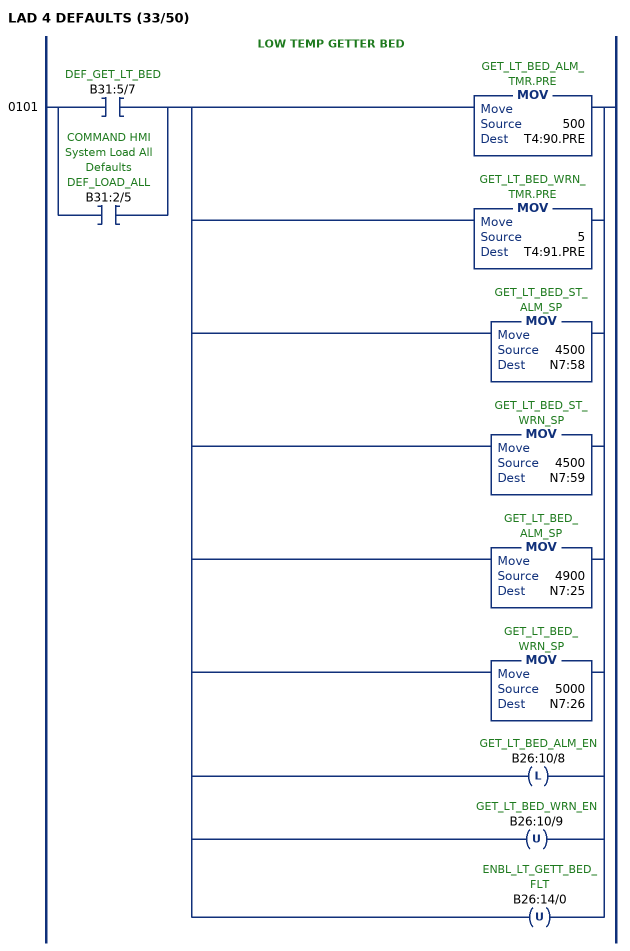
% Rung: 101 %
% TITLE: LOW TEMP GETTER BED %
SOR BST XIC B31:5/7 NXB XIC B31:2/5 BND BST MOV 500 T4:90.PRE NXB MOV 5 T4:91.PRE NXB BST MOV 4500 N7:58 NXB MOV 4500 N7:59 BND NXB BST MOV 4900 N7:25 NXB MOV 5000 N7:26 BND NXB OTL B26:10/8 NXB OTU B26:10/9 NXB OTU B26:14/0 BND EOR
%   B31:5/7  DEF_GET_LT_BED %
%   B31:2/5  DEF_LOAD_ALL  "COMMAND HMI System Load All Defaults" %
%   T4:90  GET_LT_BED_ALM_TMR %
%   T4:91  GET_LT_BED_WRN_TMR %
%   N7:58  GET_LT_BED_ST_ALM_SP %
%   N7:59  GET_LT_BED_ST_WRN_SP %
%   N7:25  GET_LT_BED_ALM_SP %
%   N7:26  GET_LT_BED_WRN_SP %
%   B26:10/8  GET_LT_BED_ALM_EN %
%   B26:10/9  GET_LT_BED_WRN_EN %
%   B26:14/0  ENBL_LT_GETT_BED_FLT %

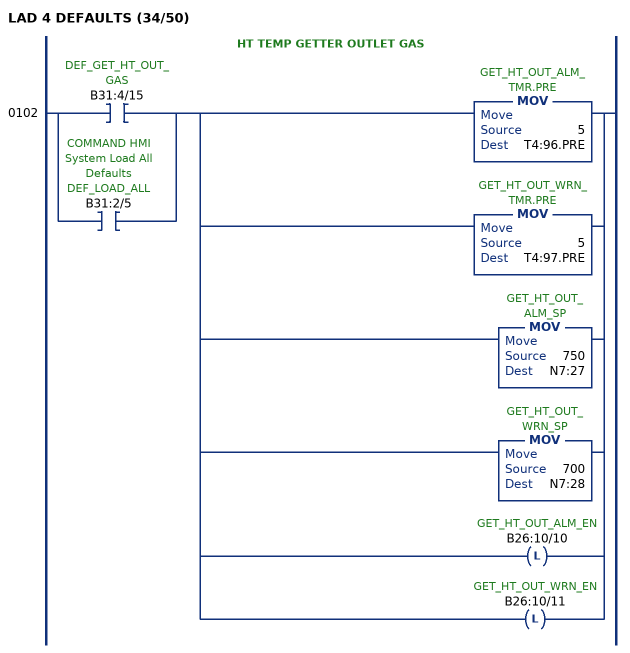
% Rung: 102 %
% TITLE: HT TEMP GETTER OUTLET GAS %
SOR BST XIC B31:4/15 NXB XIC B31:2/5 BND BST MOV 5 T4:96.PRE NXB MOV 5 T4:97.PRE NXB MOV 750 N7:27 NXB MOV 700 N7:28 NXB OTL B26:10/10 NXB OTL B26:10/11 BND EOR
%   B31:4/15  DEF_GET_HT_OUT_GAS %
%   B31:2/5  DEF_LOAD_ALL  "COMMAND HMI System Load All Defaults" %
%   T4:96  GET_HT_OUT_ALM_TMR %
%   T4:97  GET_HT_OUT_WRN_TMR %
%   N7:27  GET_HT_OUT_ALM_SP %
%   N7:28  GET_HT_OUT_WRN_SP %
%   B26:10/10  GET_HT_OUT_ALM_EN %
%   B26:10/11  GET_HT_OUT_WRN_EN %

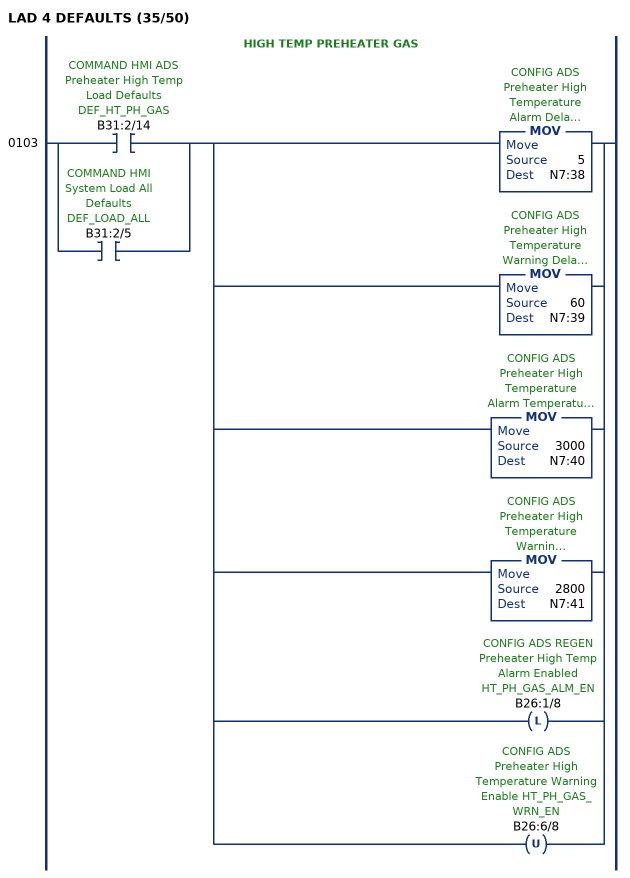
% Rung: 103 %
% TITLE: HIGH TEMP PREHEATER GAS %
SOR BST XIC B31:2/14 NXB XIC B31:2/5 BND BST MOV 5 N7:38 NXB MOV 60 N7:39 NXB MOV 3000 N7:40 NXB MOV 2800 N7:41 NXB OTL B26:1/8 NXB OTU B26:6/8 BND EOR
%   B31:2/14  DEF_HT_PH_GAS  "COMMAND HMI ADS Preheater High Temp Load Defaults" %
%   B31:2/5  DEF_LOAD_ALL  "COMMAND HMI System Load All Defaults" %
%   N7:38  HT_PH_GAS_ALM_DLY  "CONFIG ADS Preheater High Temperature Alarm Delay" %
%   N7:39  HT_PH_GAS_WRN_DLY  "CONFIG ADS Preheater High Temperature Warning Delay" %
%   N7:40  HT_PH_GAS_ALM_SP  "CONFIG ADS Preheater High Temperature Alarm Temperature" %
%   N7:41  HT_PH_GAS_WRN_SP  "CONFIG ADS Preheater High Temperature Warning Temperature" %
%   B26:1/8  HT_PH_GAS_ALM_EN  "CONFIG ADS REGEN Preheater High Temp Alarm Enabled" %
%   B26:6/8  HT_PH_GAS_WRN_EN  "CONFIG ADS Preheater High Temperature Warning Enable" %

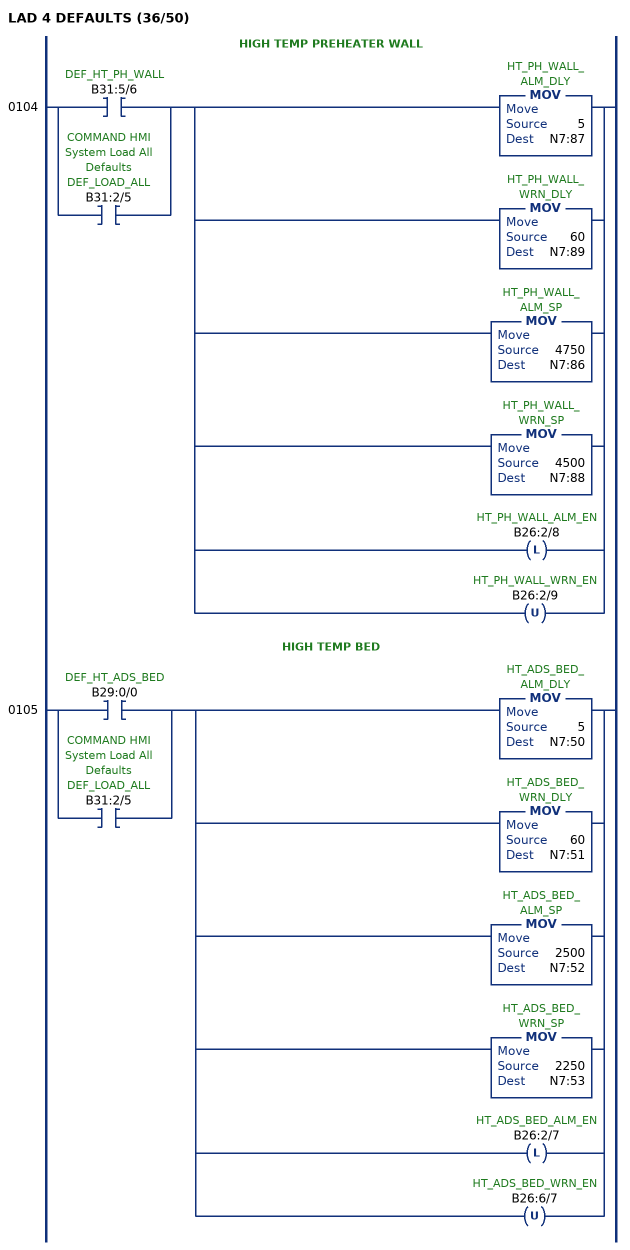
% Rung: 104 %
% TITLE: HIGH TEMP PREHEATER WALL %
SOR BST XIC B31:5/6 NXB XIC B31:2/5 BND BST MOV 5 N7:87 NXB MOV 60 N7:89 NXB MOV 4750 N7:86 NXB MOV 4500 N7:88 NXB OTL B26:2/8 NXB OTU B26:2/9 BND EOR
%   B31:5/6  DEF_HT_PH_WALL %
%   B31:2/5  DEF_LOAD_ALL  "COMMAND HMI System Load All Defaults" %
%   N7:87  HT_PH_WALL_ALM_DLY %
%   N7:89  HT_PH_WALL_WRN_DLY %
%   N7:86  HT_PH_WALL_ALM_SP %
%   N7:88  HT_PH_WALL_WRN_SP %
%   B26:2/8  HT_PH_WALL_ALM_EN %
%   B26:2/9  HT_PH_WALL_WRN_EN %
% Rung: 105 %
% TITLE: HIGH TEMP BED %
SOR BST XIC B29:0/0 NXB XIC B31:2/5 BND BST MOV 5 N7:50 NXB MOV 60 N7:51 NXB MOV 2500 N7:52 NXB MOV 2250 N7:53 NXB OTL B26:2/7 NXB OTU B26:6/7 BND EOR
%   B29:0/0  DEF_HT_ADS_BED %
%   B31:2/5  DEF_LOAD_ALL  "COMMAND HMI System Load All Defaults" %
%   N7:50  HT_ADS_BED_ALM_DLY %
%   N7:51  HT_ADS_BED_WRN_DLY %
%   N7:52  HT_ADS_BED_ALM_SP %
%   N7:53  HT_ADS_BED_WRN_SP %
%   B26:2/7  HT_ADS_BED_ALM_EN %
%   B26:6/7  HT_ADS_BED_WRN_EN %

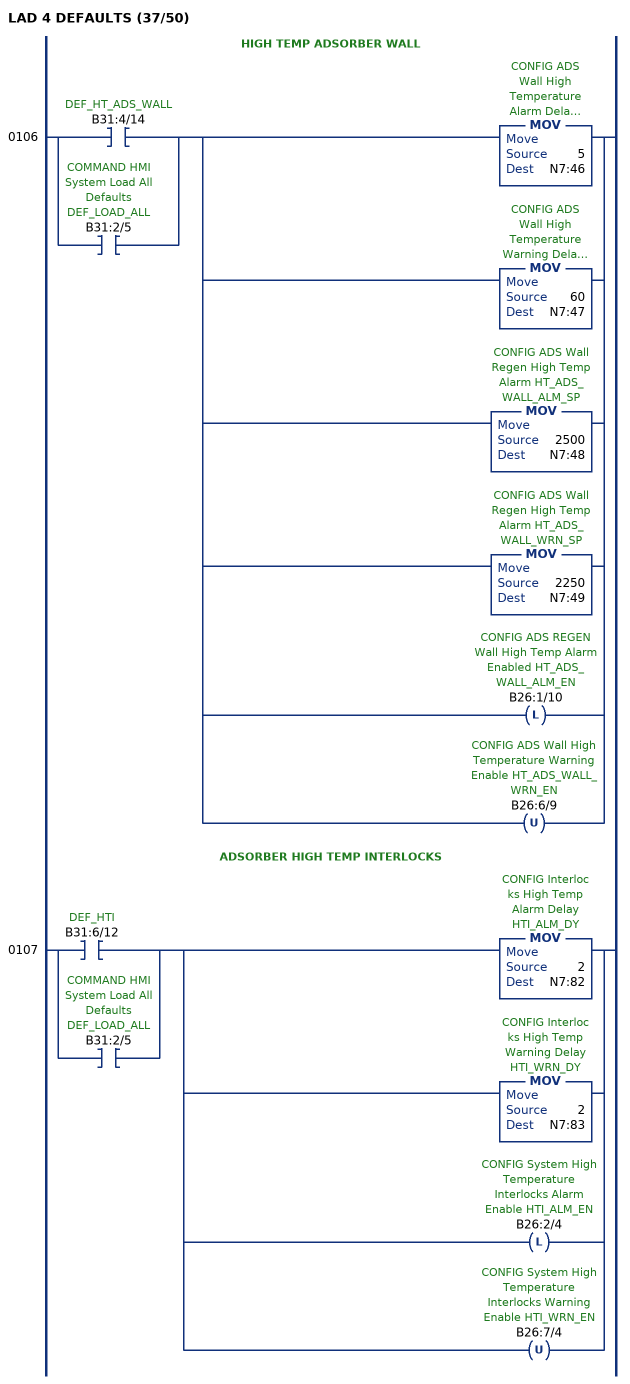
% Rung: 106 %
% TITLE: HIGH TEMP ADSORBER WALL %
SOR BST XIC B31:4/14 NXB XIC B31:2/5 BND BST MOV 5 N7:46 NXB MOV 60 N7:47 NXB MOV 2500 N7:48 NXB MOV 2250 N7:49 NXB OTL B26:1/10 NXB OTU B26:6/9 BND EOR
%   B31:4/14  DEF_HT_ADS_WALL %
%   B31:2/5  DEF_LOAD_ALL  "COMMAND HMI System Load All Defaults" %
%   N7:46  HT_ADS_WALL_ALM_DLY  "CONFIG ADS Wall High Temperature Alarm Delay" %
%   N7:47  HT_ADS_WALL_WRN_DLY  "CONFIG ADS Wall High Temperature Warning Delay" %
%   N7:48  HT_ADS_WALL_ALM_SP  "CONFIG ADS Wall Regen High Temp Alarm" %
%   N7:49  HT_ADS_WALL_WRN_SP  "CONFIG ADS Wall Regen High Temp Alarm" %
%   B26:1/10  HT_ADS_WALL_ALM_EN  "CONFIG ADS REGEN Wall High Temp Alarm Enabled" %
%   B26:6/9  HT_ADS_WALL_WRN_EN  "CONFIG ADS Wall High Temperature Warning Enable" %
% Rung: 107 %
% TITLE: ADSORBER HIGH TEMP INTERLOCKS %
SOR BST XIC B31:6/12 NXB XIC B31:2/5 BND BST MOV 2 N7:82 NXB MOV 2 N7:83 NXB OTL B26:2/4 NXB OTU B26:7/4 BND EOR
%   B31:6/12  DEF_HTI %
%   B31:2/5  DEF_LOAD_ALL  "COMMAND HMI System Load All Defaults" %
%   N7:82  HTI_ALM_DY  "CONFIG Interlocks High Temp Alarm Delay" %
%   N7:83  HTI_WRN_DY  "CONFIG Interlocks High Temp Warning Delay" %
%   B26:2/4  HTI_ALM_EN  "CONFIG System High Temperature Interlocks Alarm Enable" %
%   B26:7/4  HTI_WRN_EN  "CONFIG System High Temperature Interlocks Warning Enable" %

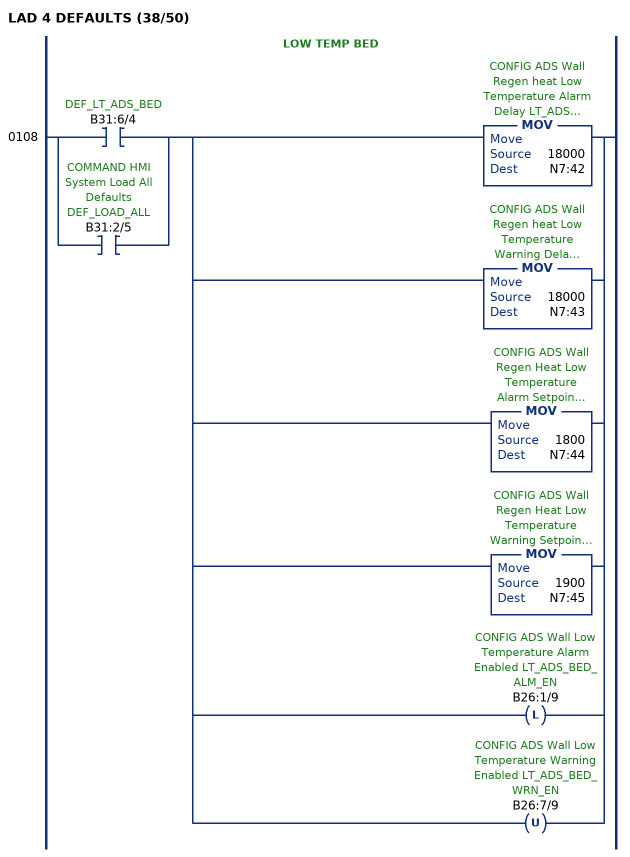
% Rung: 108 %
% TITLE: LOW TEMP BED %
SOR BST XIC B31:6/4 NXB XIC B31:2/5 BND BST MOV 18000 N7:42 NXB MOV 18000 N7:43 NXB MOV 1800 N7:44 NXB MOV 1900 N7:45 NXB OTL B26:1/9 NXB OTU B26:7/9 BND EOR
%   B31:6/4  DEF_LT_ADS_BED %
%   B31:2/5  DEF_LOAD_ALL  "COMMAND HMI System Load All Defaults" %
%   N7:42  LT_ADS_BED_ALM_DLY  "CONFIG ADS Wall Regen heat Low Temperature Alarm Delay" %
%   N7:43  LT_ADS_BED_WRN_DLY  "CONFIG ADS Wall Regen heat Low Temperature Warning Delay" %
%   N7:44  LT_ADS_BED_ALM_SP  "CONFIG ADS Wall Regen Heat Low Temperature Alarm Setpoint" %
%   N7:45  LT_ADS_BED_WRN_SP  "CONFIG ADS Wall Regen Heat Low Temperature Warning Setpoint" %
%   B26:1/9  LT_ADS_BED_ALM_EN  "CONFIG ADS Wall Low Temperature Alarm Enabled" %
%   B26:7/9  LT_ADS_BED_WRN_EN  "CONFIG ADS Wall Low Temperature Warning Enabled" %

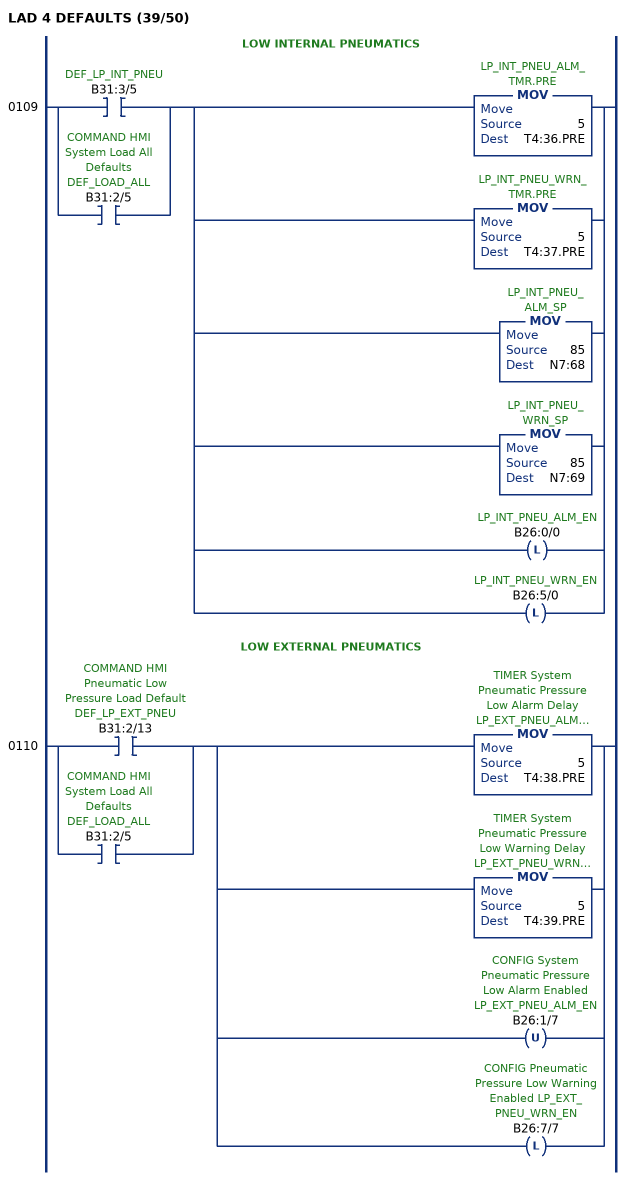
% Rung: 109 %
% TITLE: LOW INTERNAL PNEUMATICS %
SOR BST XIC B31:3/5 NXB XIC B31:2/5 BND BST MOV 5 T4:36.PRE NXB MOV 5 T4:37.PRE NXB MOV 85 N7:68 NXB MOV 85 N7:69 NXB OTL B26:0/0 NXB OTL B26:5/0 BND EOR
%   B31:3/5  DEF_LP_INT_PNEU %
%   B31:2/5  DEF_LOAD_ALL  "COMMAND HMI System Load All Defaults" %
%   T4:36  LP_INT_PNEU_ALM_TMR %
%   T4:37  LP_INT_PNEU_WRN_TMR %
%   N7:68  LP_INT_PNEU_ALM_SP %
%   N7:69  LP_INT_PNEU_WRN_SP %
%   B26:0/0  LP_INT_PNEU_ALM_EN %
%   B26:5/0  LP_INT_PNEU_WRN_EN %
% Rung: 110 %
% TITLE: LOW EXTERNAL PNEUMATICS %
SOR BST XIC B31:2/13 NXB XIC B31:2/5 BND BST MOV 5 T4:38.PRE NXB MOV 5 T4:39.PRE NXB OTU B26:1/7 NXB OTL B26:7/7 BND EOR
%   B31:2/13  DEF_LP_EXT_PNEU  "COMMAND HMI Pneumatic Low Pressure Load Default" %
%   B31:2/5  DEF_LOAD_ALL  "COMMAND HMI System Load All Defaults" %
%   T4:38  LP_EXT_PNEU_ALM_TMR  "TIMER System Pneumatic Pressure Low Alarm Delay" %
%   T4:39  LP_EXT_PNEU_WRN_TMR  "TIMER System Pneumatic Pressure Low Warning Delay" %
%   B26:1/7  LP_EXT_PNEU_ALM_EN  "CONFIG System Pneumatic Pressure Low Alarm Enabled" %
%   B26:7/7  LP_EXT_PNEU_WRN_EN  "CONFIG Pneumatic Pressure Low Warning Enabled" %

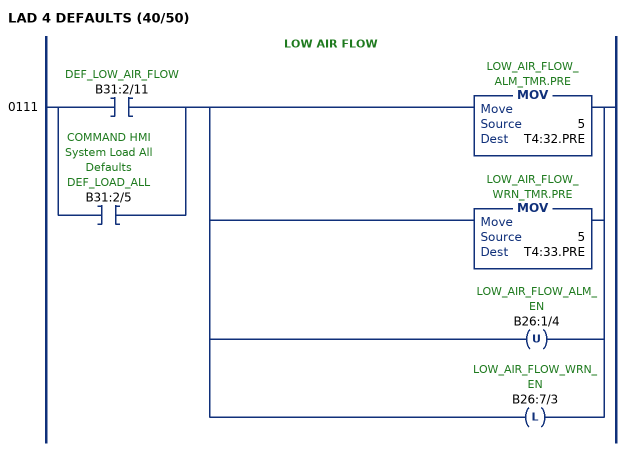
% Rung: 111 %
% TITLE: LOW AIR FLOW %
SOR BST XIC B31:2/11 NXB XIC B31:2/5 BND BST MOV 5 T4:32.PRE NXB MOV 5 T4:33.PRE NXB OTU B26:1/4 NXB OTL B26:7/3 BND EOR
%   B31:2/11  DEF_LOW_AIR_FLOW %
%   B31:2/5  DEF_LOAD_ALL  "COMMAND HMI System Load All Defaults" %
%   T4:32  LOW_AIR_FLOW_ALM_TMR %
%   T4:33  LOW_AIR_FLOW_WRN_TMR %
%   B26:1/4  LOW_AIR_FLOW_ALM_EN %
%   B26:7/3  LOW_AIR_FLOW_WRN_EN %

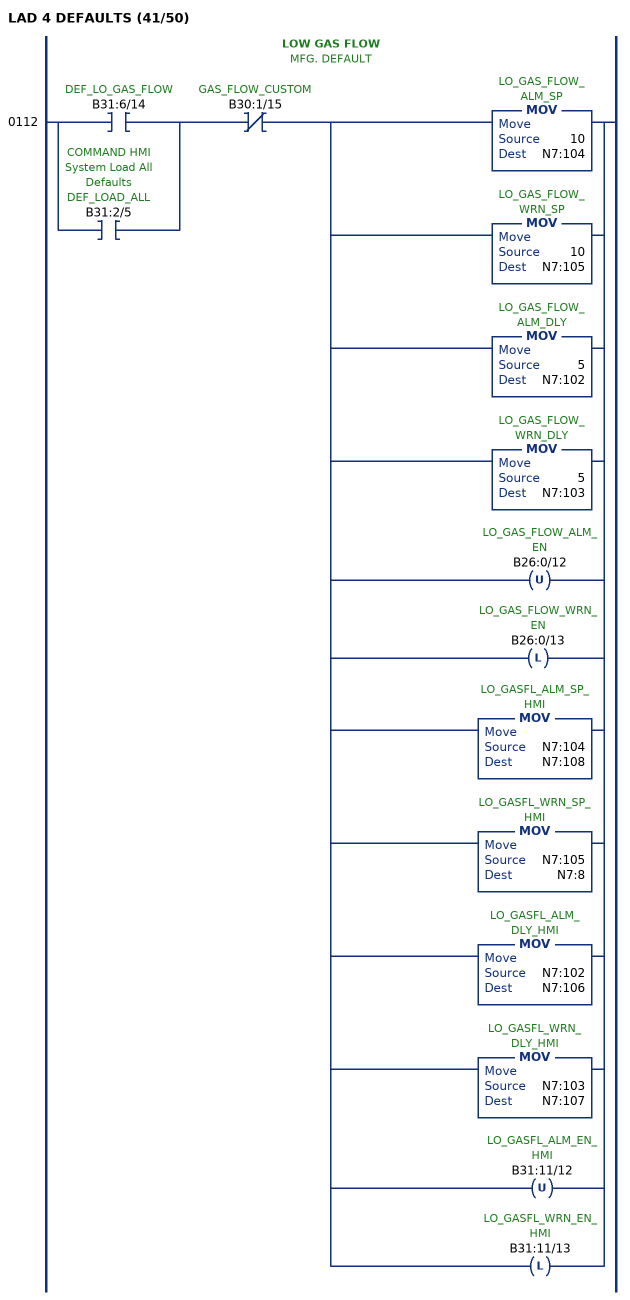
% Rung: 112 %
% TITLE: LOW GAS FLOW %
% MFG. DEFAULT %
SOR BST XIC B31:6/14 NXB XIC B31:2/5 BND XIO B30:1/15 BST MOV 10 N7:104 NXB MOV 10 N7:105 NXB MOV 5 N7:102 NXB MOV 5 N7:103 NXB OTU B26:0/12 NXB OTL B26:0/13 NXB MOV N7:104 N7:108 NXB MOV N7:105 N7:8 NXB MOV N7:102 N7:106 NXB MOV N7:103 N7:107 NXB OTU B31:11/12 NXB OTL B31:11/13 BND EOR
%   B31:6/14  DEF_LO_GAS_FLOW %
%   B31:2/5  DEF_LOAD_ALL  "COMMAND HMI System Load All Defaults" %
%   B30:1/15  GAS_FLOW_CUSTOM %
%   N7:104  LO_GAS_FLOW_ALM_SP %
%   N7:105  LO_GAS_FLOW_WRN_SP %
%   N7:102  LO_GAS_FLOW_ALM_DLY %
%   N7:103  LO_GAS_FLOW_WRN_DLY %
%   B26:0/12  LO_GAS_FLOW_ALM_EN %
%   B26:0/13  LO_GAS_FLOW_WRN_EN %
%   N7:108  LO_GASFL_ALM_SP_HMI %
%   N7:8  LO_GASFL_WRN_SP_HMI %
%   N7:106  LO_GASFL_ALM_DLY_HMI %
%   N7:107  LO_GASFL_WRN_DLY_HMI %
%   B31:11/12  LO_GASFL_ALM_EN_HMI %
%   B31:11/13  LO_GASFL_WRN_EN_HMI %

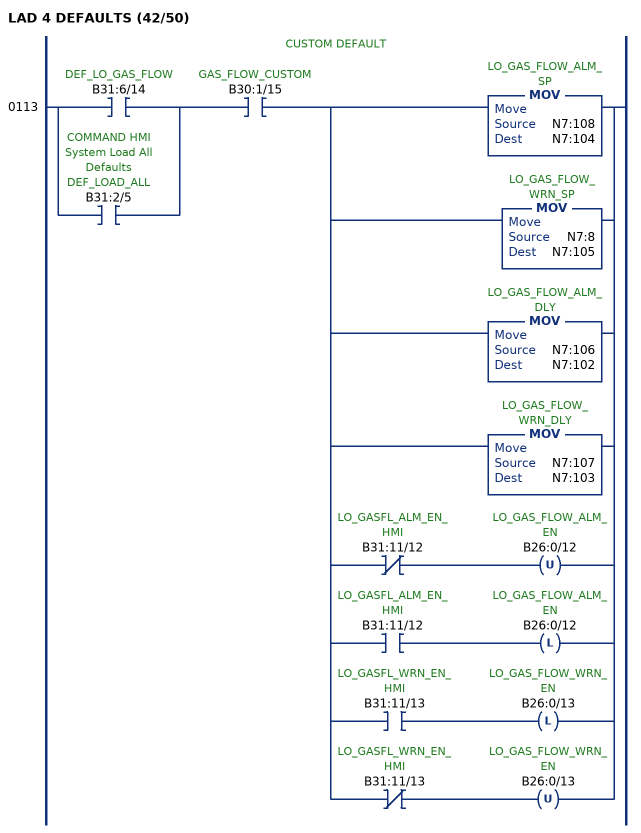
% Rung: 113 %
% CUSTOM DEFAULT %
SOR BST XIC B31:6/14 NXB XIC B31:2/5 BND XIC B30:1/15 BST MOV N7:108 N7:104 NXB MOV N7:8 N7:105 NXB MOV N7:106 N7:102 NXB MOV N7:107 N7:103 NXB XIO B31:11/12 OTU B26:0/12 NXB XIC B31:11/12 OTL B26:0/12 NXB XIC B31:11/13 OTL B26:0/13 NXB XIO B31:11/13 OTU B26:0/13 BND EOR
%   B31:6/14  DEF_LO_GAS_FLOW %
%   B31:2/5  DEF_LOAD_ALL  "COMMAND HMI System Load All Defaults" %
%   B30:1/15  GAS_FLOW_CUSTOM %
%   N7:108  LO_GASFL_ALM_SP_HMI %
%   N7:104  LO_GAS_FLOW_ALM_SP %
%   N7:8  LO_GASFL_WRN_SP_HMI %
%   N7:105  LO_GAS_FLOW_WRN_SP %
%   N7:106  LO_GASFL_ALM_DLY_HMI %
%   N7:102  LO_GAS_FLOW_ALM_DLY %
%   N7:107  LO_GASFL_WRN_DLY_HMI %
%   N7:103  LO_GAS_FLOW_WRN_DLY %
%   B31:11/12  LO_GASFL_ALM_EN_HMI %
%   B26:0/12  LO_GAS_FLOW_ALM_EN %
%   B31:11/13  LO_GASFL_WRN_EN_HMI %
%   B26:0/13  LO_GAS_FLOW_WRN_EN %

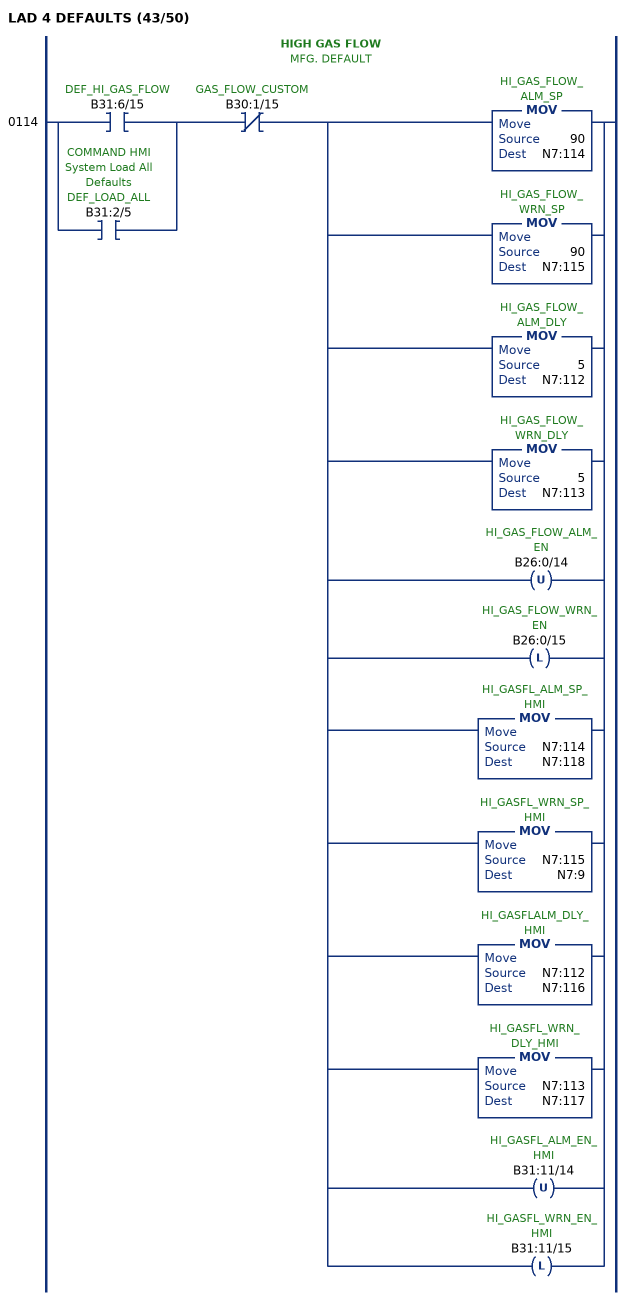
% Rung: 114 %
% TITLE: HIGH GAS FLOW %
% MFG. DEFAULT %
SOR BST XIC B31:6/15 NXB XIC B31:2/5 BND XIO B30:1/15 BST MOV 90 N7:114 NXB MOV 90 N7:115 NXB MOV 5 N7:112 NXB MOV 5 N7:113 NXB OTU B26:0/14 NXB OTL B26:0/15 NXB MOV N7:114 N7:118 NXB MOV N7:115 N7:9 NXB MOV N7:112 N7:116 NXB MOV N7:113 N7:117 NXB OTU B31:11/14 NXB OTL B31:11/15 BND EOR
%   B31:6/15  DEF_HI_GAS_FLOW %
%   B31:2/5  DEF_LOAD_ALL  "COMMAND HMI System Load All Defaults" %
%   B30:1/15  GAS_FLOW_CUSTOM %
%   N7:114  HI_GAS_FLOW_ALM_SP %
%   N7:115  HI_GAS_FLOW_WRN_SP %
%   N7:112  HI_GAS_FLOW_ALM_DLY %
%   N7:113  HI_GAS_FLOW_WRN_DLY %
%   B26:0/14  HI_GAS_FLOW_ALM_EN %
%   B26:0/15  HI_GAS_FLOW_WRN_EN %
%   N7:118  HI_GASFL_ALM_SP_HMI %
%   N7:9  HI_GASFL_WRN_SP_HMI %
%   N7:116  HI_GASFLALM_DLY_HMI %
%   N7:117  HI_GASFL_WRN_DLY_HMI %
%   B31:11/14  HI_GASFL_ALM_EN_HMI %
%   B31:11/15  HI_GASFL_WRN_EN_HMI %

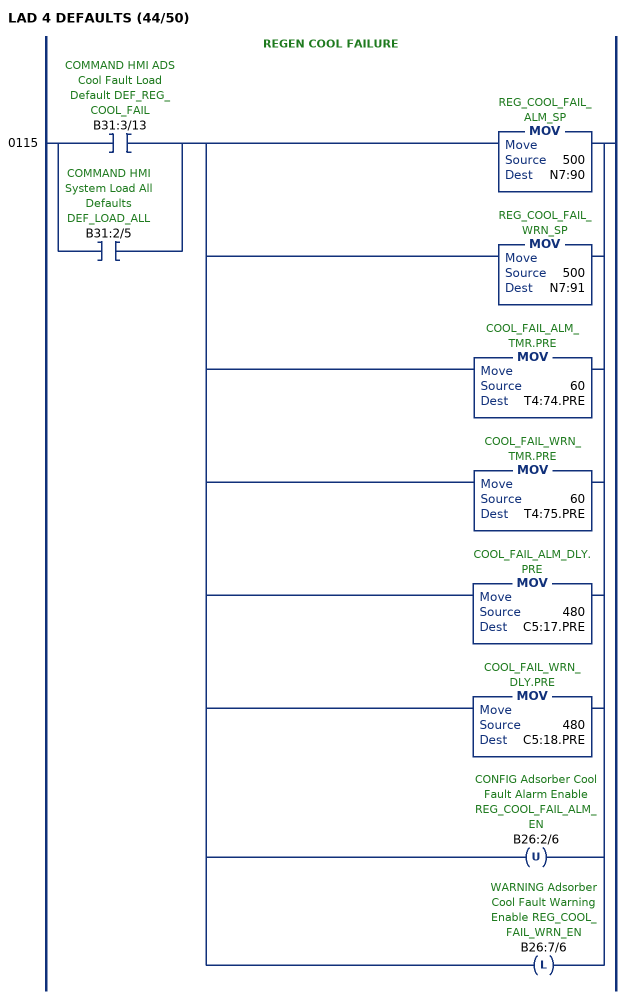
% Rung: 115 %
% TITLE: REGEN COOL FAILURE %
SOR BST XIC B31:3/13 NXB XIC B31:2/5 BND BST MOV 500 N7:90 NXB MOV 500 N7:91 NXB MOV 60 T4:74.PRE NXB MOV 60 T4:75.PRE NXB MOV 480 C5:17.PRE NXB MOV 480 C5:18.PRE NXB OTU B26:2/6 NXB OTL B26:7/6 BND EOR
%   B31:3/13  DEF_REG_COOL_FAIL  "COMMAND HMI ADS Cool Fault Load Default" %
%   B31:2/5  DEF_LOAD_ALL  "COMMAND HMI System Load All Defaults" %
%   N7:90  REG_COOL_FAIL_ALM_SP %
%   N7:91  REG_COOL_FAIL_WRN_SP %
%   T4:74  COOL_FAIL_ALM_TMR %
%   T4:75  COOL_FAIL_WRN_TMR %
%   C5:17  COOL_FAIL_ALM_DLY %
%   C5:18  COOL_FAIL_WRN_DLY %
%   B26:2/6  REG_COOL_FAIL_ALM_EN  "CONFIG Adsorber Cool Fault Alarm Enable" %
%   B26:7/6  REG_COOL_FAIL_WRN_EN  "WARNING Adsorber Cool Fault Warning Enable" %

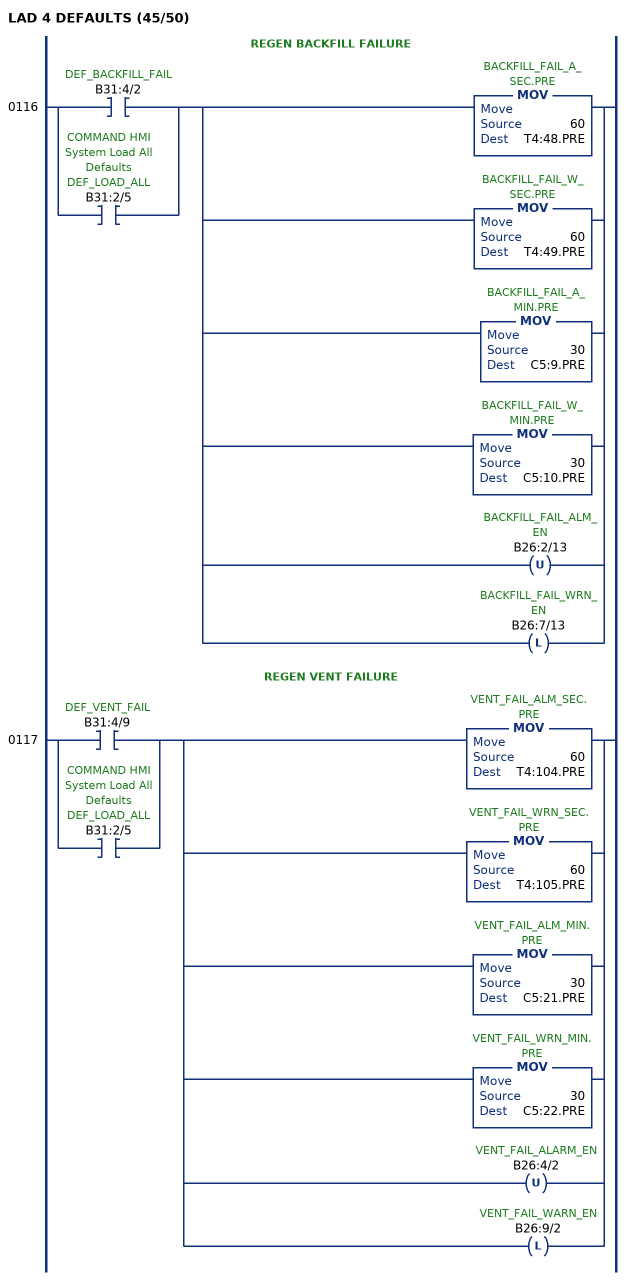
% Rung: 116 %
% TITLE: REGEN BACKFILL FAILURE %
SOR BST XIC B31:4/2 NXB XIC B31:2/5 BND BST MOV 60 T4:48.PRE NXB MOV 60 T4:49.PRE NXB MOV 30 C5:9.PRE NXB MOV 30 C5:10.PRE NXB OTU B26:2/13 NXB OTL B26:7/13 BND EOR
%   B31:4/2  DEF_BACKFILL_FAIL %
%   B31:2/5  DEF_LOAD_ALL  "COMMAND HMI System Load All Defaults" %
%   T4:48  BACKFILL_FAIL_A_SEC %
%   T4:49  BACKFILL_FAIL_W_SEC %
%   C5:9  BACKFILL_FAIL_A_MIN %
%   C5:10  BACKFILL_FAIL_W_MIN %
%   B26:2/13  BACKFILL_FAIL_ALM_EN %
%   B26:7/13  BACKFILL_FAIL_WRN_EN %
% Rung: 117 %
% TITLE: REGEN VENT FAILURE %
SOR BST XIC B31:4/9 NXB XIC B31:2/5 BND BST MOV 60 T4:104.PRE NXB MOV 60 T4:105.PRE NXB MOV 30 C5:21.PRE NXB MOV 30 C5:22.PRE NXB OTU B26:4/2 NXB OTL B26:9/2 BND EOR
%   B31:4/9  DEF_VENT_FAIL %
%   B31:2/5  DEF_LOAD_ALL  "COMMAND HMI System Load All Defaults" %
%   T4:104  VENT_FAIL_ALM_SEC %
%   T4:105  VENT_FAIL_WRN_SEC %
%   C5:21  VENT_FAIL_ALM_MIN %
%   C5:22  VENT_FAIL_WRN_MIN %
%   B26:4/2  VENT_FAIL_ALARM_EN %
%   B26:9/2  VENT_FAIL_WARN_EN %

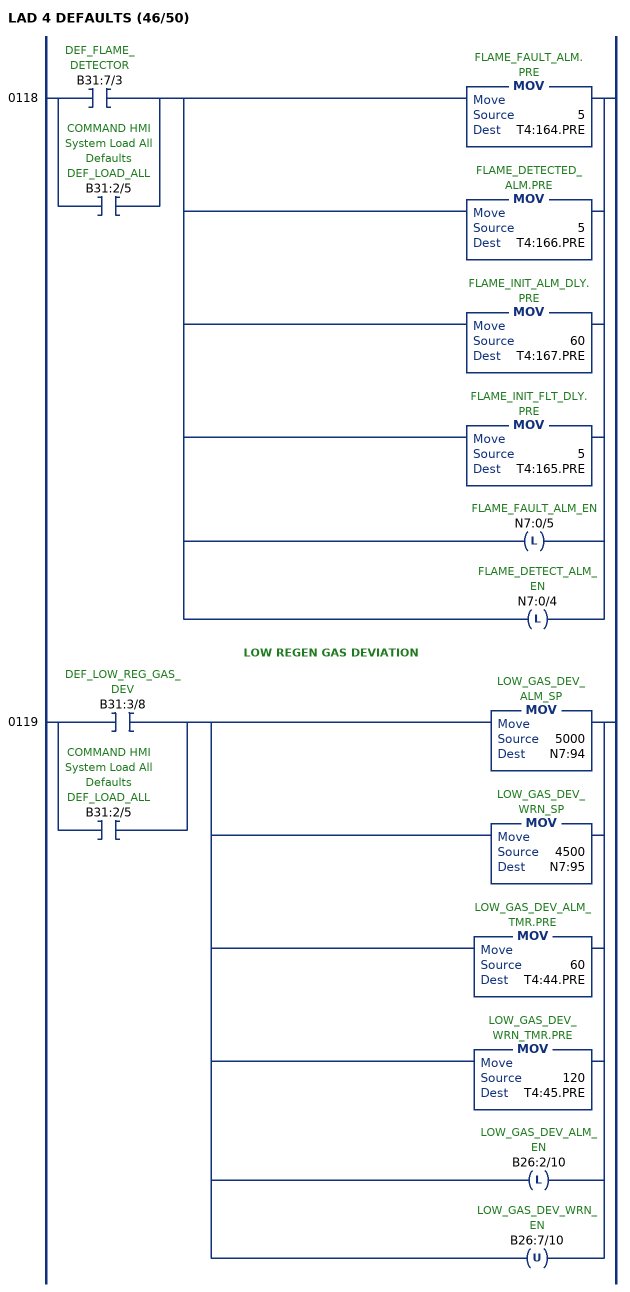
% Rung: 118 %
SOR BST XIC B31:7/3 NXB XIC B31:2/5 BND BST MOV 5 T4:164.PRE NXB MOV 5 T4:166.PRE NXB MOV 60 T4:167.PRE NXB MOV 5 T4:165.PRE NXB OTL N7:0/5 NXB OTL N7:0/4 BND EOR
%   B31:7/3  DEF_FLAME_DETECTOR %
%   B31:2/5  DEF_LOAD_ALL  "COMMAND HMI System Load All Defaults" %
%   T4:164  FLAME_FAULT_ALM %
%   T4:166  FLAME_DETECTED_ALM %
%   T4:167  FLAME_INIT_ALM_DLY %
%   T4:165  FLAME_INIT_FLT_DLY %
%   N7:0/5  FLAME_FAULT_ALM_EN %
%   N7:0/4  FLAME_DETECT_ALM_EN %
% Rung: 119 %
% TITLE: LOW REGEN GAS DEVIATION %
SOR BST XIC B31:3/8 NXB XIC B31:2/5 BND BST MOV 5000 N7:94 NXB MOV 4500 N7:95 NXB MOV 60 T4:44.PRE NXB MOV 120 T4:45.PRE NXB OTL B26:2/10 NXB OTU B26:7/10 BND EOR
%   B31:3/8  DEF_LOW_REG_GAS_DEV %
%   B31:2/5  DEF_LOAD_ALL  "COMMAND HMI System Load All Defaults" %
%   N7:94  LOW_GAS_DEV_ALM_SP %
%   N7:95  LOW_GAS_DEV_WRN_SP %
%   T4:44  LOW_GAS_DEV_ALM_TMR %
%   T4:45  LOW_GAS_DEV_WRN_TMR %
%   B26:2/10  LOW_GAS_DEV_ALM_EN %
%   B26:7/10  LOW_GAS_DEV_WRN_EN %

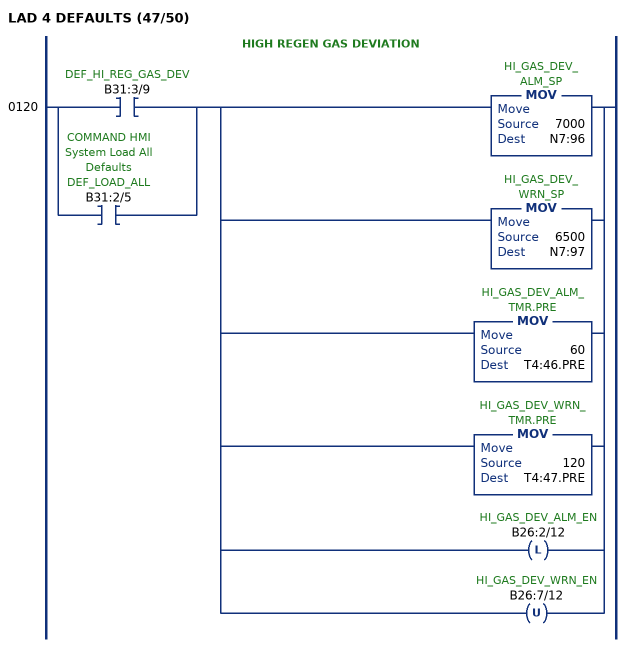
% Rung: 120 %
% TITLE: HIGH REGEN GAS DEVIATION %
SOR BST XIC B31:3/9 NXB XIC B31:2/5 BND BST MOV 7000 N7:96 NXB MOV 6500 N7:97 NXB MOV 60 T4:46.PRE NXB MOV 120 T4:47.PRE NXB OTL B26:2/12 NXB OTU B26:7/12 BND EOR
%   B31:3/9  DEF_HI_REG_GAS_DEV %
%   B31:2/5  DEF_LOAD_ALL  "COMMAND HMI System Load All Defaults" %
%   N7:96  HI_GAS_DEV_ALM_SP %
%   N7:97  HI_GAS_DEV_WRN_SP %
%   T4:46  HI_GAS_DEV_ALM_TMR %
%   T4:47  HI_GAS_DEV_WRN_TMR %
%   B26:2/12  HI_GAS_DEV_ALM_EN %
%   B26:7/12  HI_GAS_DEV_WRN_EN %

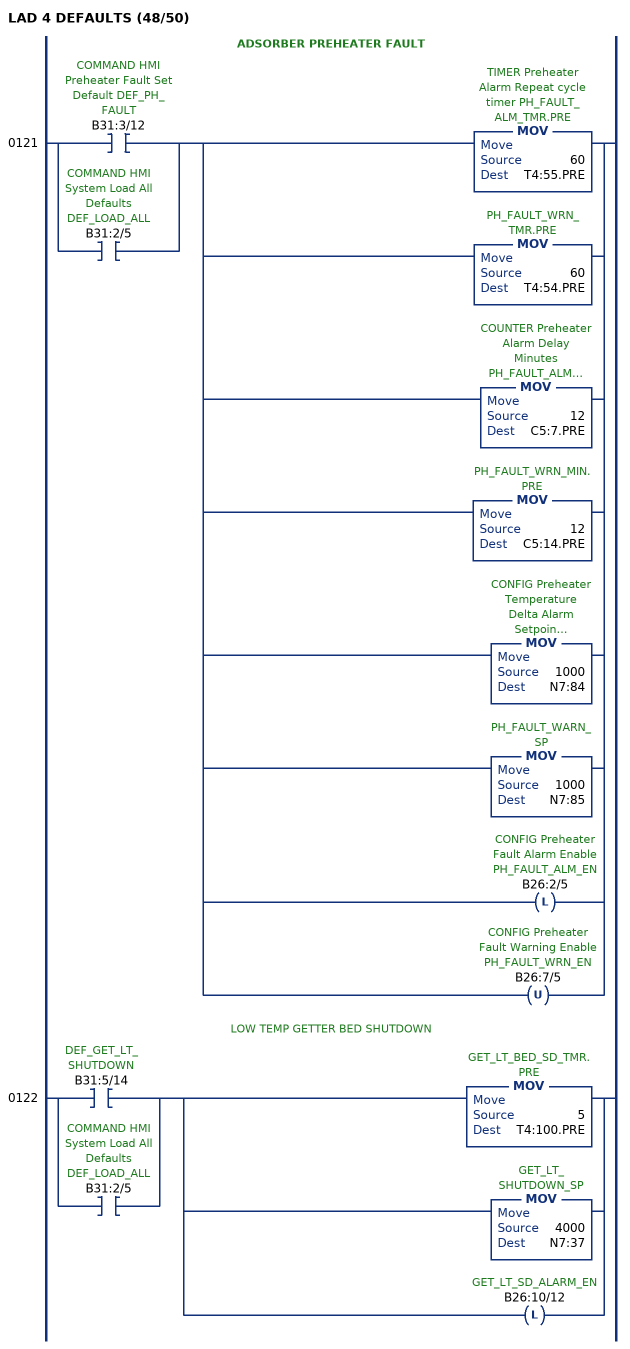
% Rung: 121 %
% TITLE: ADSORBER PREHEATER FAULT %
SOR BST XIC B31:3/12 NXB XIC B31:2/5 BND BST MOV 60 T4:55.PRE NXB MOV 60 T4:54.PRE NXB MOV 12 C5:7.PRE NXB MOV 12 C5:14.PRE NXB MOV 1000 N7:84 NXB MOV 1000 N7:85 NXB OTL B26:2/5 NXB OTU B26:7/5 BND EOR
%   B31:3/12  DEF_PH_FAULT  "COMMAND HMI Preheater Fault Set Default" %
%   B31:2/5  DEF_LOAD_ALL  "COMMAND HMI System Load All Defaults" %
%   T4:55  PH_FAULT_ALM_TMR  "TIMER Preheater Alarm Repeat cycle timer" %
%   T4:54  PH_FAULT_WRN_TMR %
%   C5:7  PH_FAULT_ALM_MIN  "COUNTER Preheater Alarm Delay Minutes" %
%   C5:14  PH_FAULT_WRN_MIN %
%   N7:84  PH_FAULT_ALARM_SP  "CONFIG Preheater Temperature Delta Alarm Setpoint" %
%   N7:85  PH_FAULT_WARN_SP %
%   B26:2/5  PH_FAULT_ALM_EN  "CONFIG Preheater Fault Alarm Enable" %
%   B26:7/5  PH_FAULT_WRN_EN  "CONFIG Preheater Fault Warning Enable" %
% Rung: 122 %
% LOW TEMP GETTER BED SHUTDOWN %
SOR BST XIC B31:5/14 NXB XIC B31:2/5 BND BST MOV 5 T4:100.PRE NXB MOV 4000 N7:37 NXB OTL B26:10/12 BND EOR
%   B31:5/14  DEF_GET_LT_SHUTDOWN %
%   B31:2/5  DEF_LOAD_ALL  "COMMAND HMI System Load All Defaults" %
%   T4:100  GET_LT_BED_SD_TMR %
%   N7:37  GET_LT_SHUTDOWN_SP %
%   B26:10/12  GET_LT_SD_ALARM_EN %

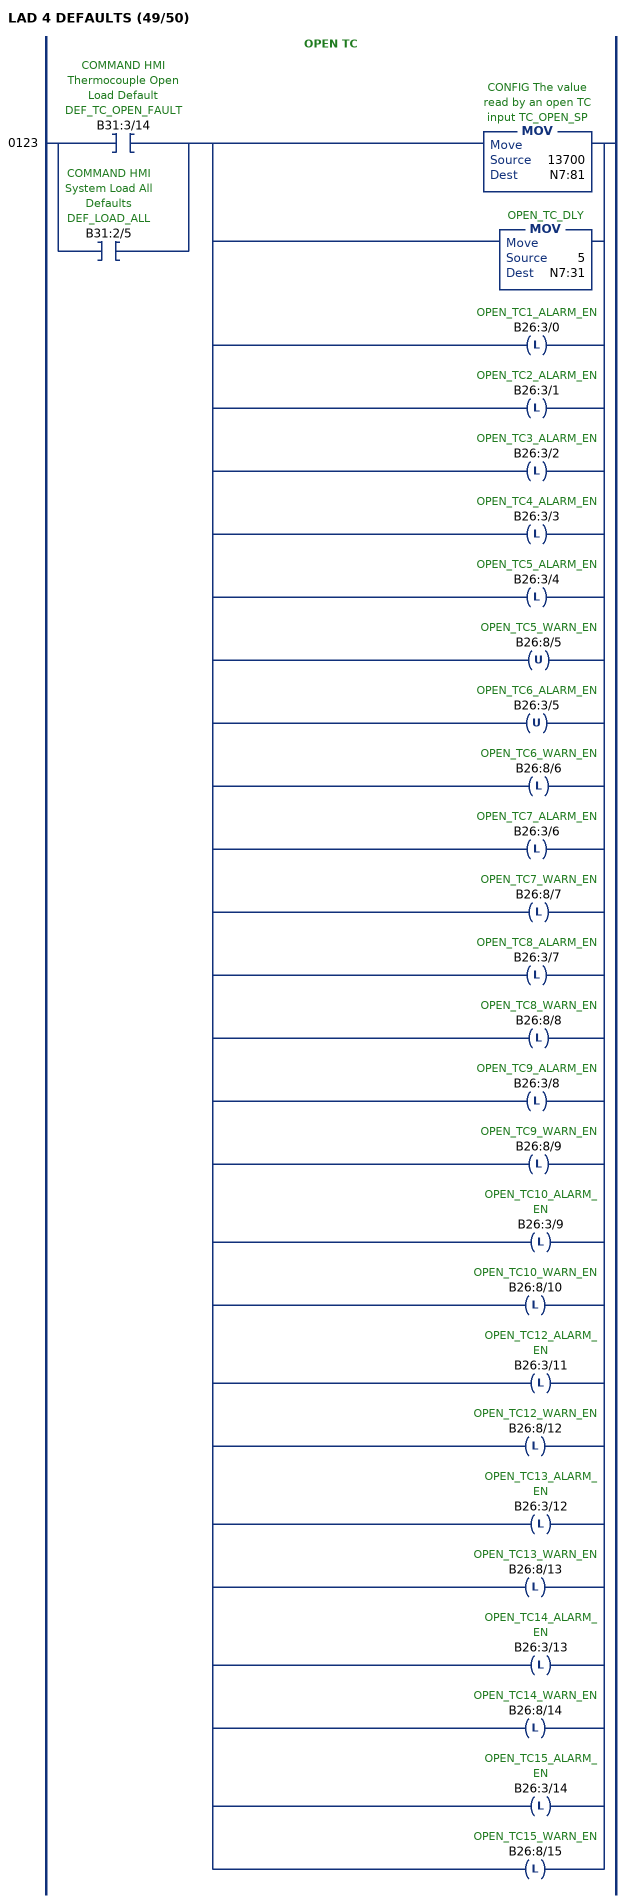
% Rung: 123 %
% TITLE: OPEN TC %
SOR BST XIC B31:3/14 NXB XIC B31:2/5 BND BST MOV 13700 N7:81 NXB MOV 5 N7:31 NXB OTL B26:3/0 NXB OTL B26:3/1 NXB OTL B26:3/2 NXB OTL B26:3/3 NXB OTL B26:3/4 NXB OTU B26:8/5 NXB OTU B26:3/5 NXB OTL B26:8/6 NXB OTL B26:3/6 NXB OTL B26:8/7 NXB OTL B26:3/7 NXB OTL B26:8/8 NXB OTL B26:3/8 NXB OTL B26:8/9 NXB OTL B26:3/9 NXB OTL B26:8/10 NXB OTL B26:3/11 NXB OTL B26:8/12 NXB OTL B26:3/12 NXB OTL B26:8/13 NXB OTL B26:3/13 NXB OTL B26:8/14 NXB OTL B26:3/14 NXB OTL B26:8/15 BND EOR
%   B31:3/14  DEF_TC_OPEN_FAULT  "COMMAND HMI Thermocouple Open Load Default" %
%   B31:2/5  DEF_LOAD_ALL  "COMMAND HMI System Load All Defaults" %
%   N7:81  TC_OPEN_SP  "CONFIG The value read by an open TC input" %
%   N7:31  OPEN_TC_DLY %
%   B26:3/0  OPEN_TC1_ALARM_EN %
%   B26:3/1  OPEN_TC2_ALARM_EN %
%   B26:3/2  OPEN_TC3_ALARM_EN %
%   B26:3/3  OPEN_TC4_ALARM_EN %
%   B26:3/4  OPEN_TC5_ALARM_EN %
%   B26:8/5  OPEN_TC5_WARN_EN %
%   B26:3/5  OPEN_TC6_ALARM_EN %
%   B26:8/6  OPEN_TC6_WARN_EN %
%   B26:3/6  OPEN_TC7_ALARM_EN %
%   B26:8/7  OPEN_TC7_WARN_EN %
%   B26:3/7  OPEN_TC8_ALARM_EN %
%   B26:8/8  OPEN_TC8_WARN_EN %
%   B26:3/8  OPEN_TC9_ALARM_EN %
%   B26:8/9  OPEN_TC9_WARN_EN %
%   B26:3/9  OPEN_TC10_ALARM_EN %
%   B26:8/10  OPEN_TC10_WARN_EN %
%   B26:3/11  OPEN_TC12_ALARM_EN %
%   B26:8/12  OPEN_TC12_WARN_EN %
%   B26:3/12  OPEN_TC13_ALARM_EN %
%   B26:8/13  OPEN_TC13_WARN_EN %
%   B26:3/13  OPEN_TC14_ALARM_EN %
%   B26:8/14  OPEN_TC14_WARN_EN %
%   B26:3/14  OPEN_TC15_ALARM_EN %
%   B26:8/15  OPEN_TC15_WARN_EN %

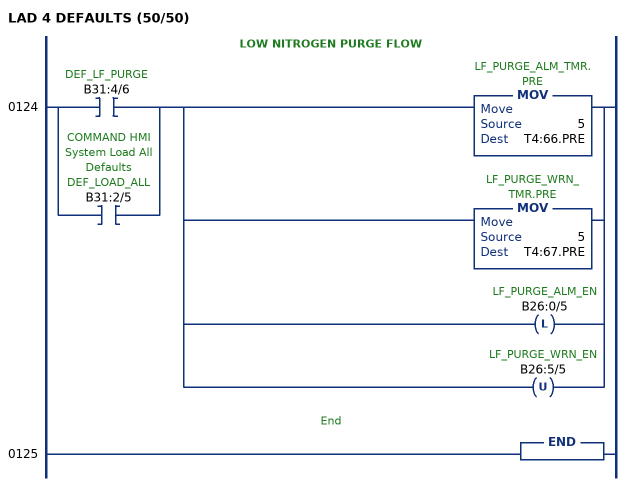
% Rung: 124 %
% TITLE: LOW NITROGEN PURGE FLOW %
SOR BST XIC B31:4/6 NXB XIC B31:2/5 BND BST MOV 5 T4:66.PRE NXB MOV 5 T4:67.PRE NXB OTL B26:0/5 NXB OTU B26:5/5 BND EOR
%   B31:4/6  DEF_LF_PURGE %
%   B31:2/5  DEF_LOAD_ALL  "COMMAND HMI System Load All Defaults" %
%   T4:66  LF_PURGE_ALM_TMR %
%   T4:67  LF_PURGE_WRN_TMR %
%   B26:0/5  LF_PURGE_ALM_EN %
%   B26:5/5  LF_PURGE_WRN_EN %
% Rung: 125 %
% End %
SOR END EOR

LADDER 5 "SYS_FAULTS"    % Monitors the system fault conditions %
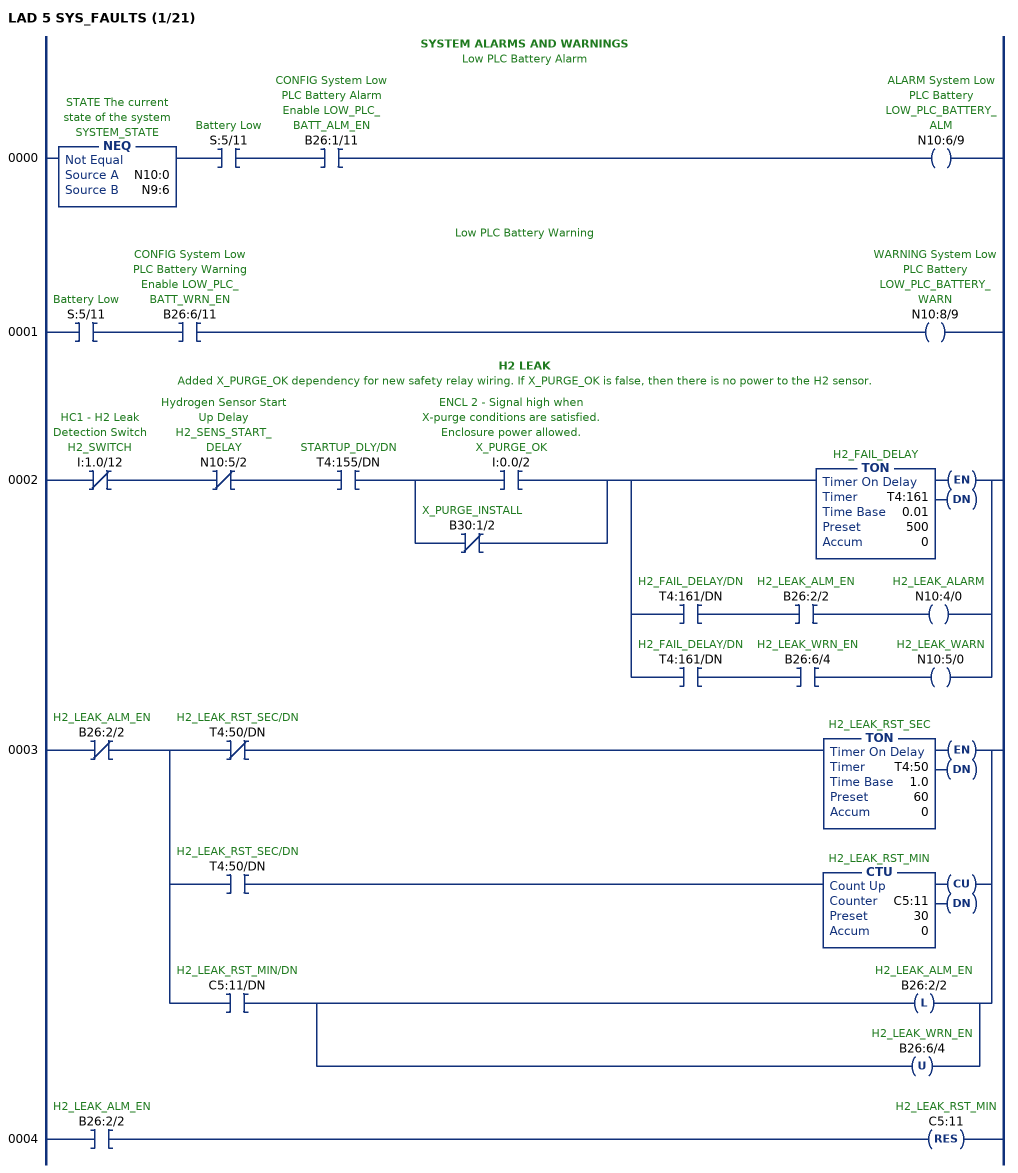
% Rung: 0 %
% TITLE: SYSTEM ALARMS AND WARNINGS %
% Low PLC Battery Alarm %
SOR NEQ N10:0 N9:6 XIC S:5/11 XIC B26:1/11 OTE N10:6/9 EOR
%   N10:0  SYSTEM_STATE  "STATE The current state of the system" %
%   N9:6  SYSTEM_PURGE %
%   S:5/11  "Battery Low" %
%   B26:1/11  LOW_PLC_BATT_ALM_EN  "CONFIG System Low PLC Battery Alarm Enable" %
%   N10:6/9  LOW_PLC_BATTERY_ALM  "ALARM System Low PLC Battery" %
% Rung: 1 %
% Low PLC Battery Warning %
SOR XIC S:5/11 XIC B26:6/11 OTE N10:8/9 EOR
%   S:5/11  "Battery Low" %
%   B26:6/11  LOW_PLC_BATT_WRN_EN  "CONFIG System Low PLC Battery Warning Enable" %
%   N10:8/9  LOW_PLC_BATTERY_WARN  "WARNING System Low PLC Battery" %
% Rung: 2 %
% TITLE: H2 LEAK %
% Added X_PURGE_OK dependency for new safety relay wiring. If X_PURGE_OK is false, then there is no power to the H2 sensor. %
SOR XIO I:1.0/12 XIO N10:5/2 XIC T4:155/DN BST XIC I:0.0/2 NXB XIO B30:1/2 BND BST TON T4:161 0.01 500 0 NXB XIC T4:161/DN XIC B26:2/2 OTE N10:4/0 NXB XIC T4:161/DN XIC B26:6/4 OTE N10:5/0 BND EOR
%   I:1.0/12  H2_SWITCH  "HC1 - H2 Leak Detection Switch" %
%   N10:5/2  H2_SENS_START_DELAY  "Hydrogen Sensor Start Up Delay" %
%   T4:155  STARTUP_DLY %
%   I:0.0/2  X_PURGE_OK  "ENCL 2 - Signal high when X-purge conditions are satisfied. Enclosure power allowed." %
%   B30:1/2  X_PURGE_INSTALL %
%   T4:161  H2_FAIL_DELAY %
%   B26:2/2  H2_LEAK_ALM_EN %
%   N10:4/0  H2_LEAK_ALARM %
%   B26:6/4  H2_LEAK_WRN_EN %
%   N10:5/0  H2_LEAK_WARN %
% Rung: 3 %
SOR XIO B26:2/2 BST XIO T4:50/DN TON T4:50 1.0 60 0 NXB XIC T4:50/DN CTU C5:11 30 0 NXB XIC C5:11/DN BST OTL B26:2/2 NXB OTU B26:6/4 BND BND EOR
%   B26:2/2  H2_LEAK_ALM_EN %
%   T4:50  H2_LEAK_RST_SEC %
%   C5:11  H2_LEAK_RST_MIN %
%   B26:6/4  H2_LEAK_WRN_EN %
% Rung: 4 %
SOR XIC B26:2/2 RES C5:11 EOR
%   B26:2/2  H2_LEAK_ALM_EN %
%   C5:11  H2_LEAK_RST_MIN %

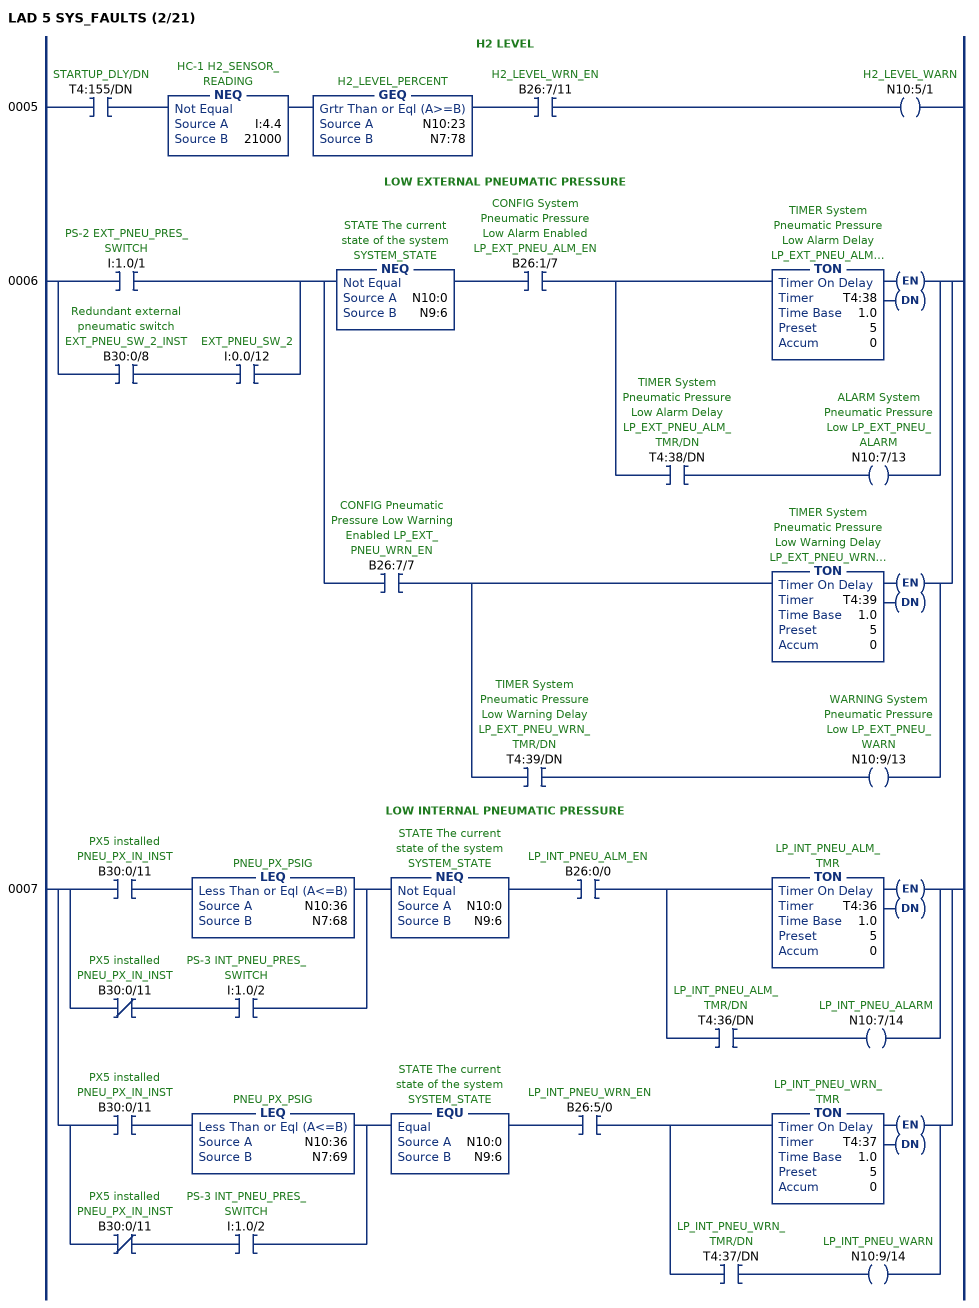
% Rung: 5 %
% TITLE: H2 LEVEL %
SOR XIC T4:155/DN NEQ I:4.4 21000 GEQ N10:23 N7:78 XIC B26:7/11 OTE N10:5/1 EOR
%   T4:155  STARTUP_DLY %
%   I:4.4  H2_SENSOR_READING  "HC-1" %
%   N10:23  H2_LEVEL_PERCENT %
%   N7:78  H2_LEVEL_WRN_SP %
%   B26:7/11  H2_LEVEL_WRN_EN %
%   N10:5/1  H2_LEVEL_WARN %
% Rung: 6 %
% TITLE: LOW EXTERNAL PNEUMATIC PRESSURE %
SOR BST XIC I:1.0/1 NXB XIC B30:0/8 XIC I:0.0/12 BND BST NEQ N10:0 N9:6 XIC B26:1/7 BST TON T4:38 1.0 5 0 NXB XIC T4:38/DN OTE N10:7/13 BND NXB XIC B26:7/7 BST TON T4:39 1.0 5 0 NXB XIC T4:39/DN OTE N10:9/13 BND BND EOR
%   I:1.0/1  EXT_PNEU_PRES_SWITCH  "PS-2" %
%   B30:0/8  EXT_PNEU_SW_2_INST  "Redundant external pneumatic switch" %
%   I:0.0/12  EXT_PNEU_SW_2 %
%   N10:0  SYSTEM_STATE  "STATE The current state of the system" %
%   N9:6  SYSTEM_PURGE %
%   B26:1/7  LP_EXT_PNEU_ALM_EN  "CONFIG System Pneumatic Pressure Low Alarm Enabled" %
%   T4:38  LP_EXT_PNEU_ALM_TMR  "TIMER System Pneumatic Pressure Low Alarm Delay" %
%   N10:7/13  LP_EXT_PNEU_ALARM  "ALARM System Pneumatic Pressure Low" %
%   B26:7/7  LP_EXT_PNEU_WRN_EN  "CONFIG Pneumatic Pressure Low Warning Enabled" %
%   T4:39  LP_EXT_PNEU_WRN_TMR  "TIMER System Pneumatic Pressure Low Warning Delay" %
%   N10:9/13  LP_EXT_PNEU_WARN  "WARNING System Pneumatic Pressure Low" %
% Rung: 7 %
% TITLE: LOW INTERNAL PNEUMATIC PRESSURE %
SOR BST BST XIC B30:0/11 LEQ N10:36 N7:68 NXB XIO B30:0/11 XIC I:1.0/2 BND NEQ N10:0 N9:6 XIC B26:0/0 BST TON T4:36 1.0 5 0 NXB XIC T4:36/DN OTE N10:7/14 BND NXB BST XIC B30:0/11 LEQ N10:36 N7:69 NXB XIO B30:0/11 XIC I:1.0/2 BND EQU N10:0 N9:6 XIC B26:5/0 BST TON T4:37 1.0 5 0 NXB XIC T4:37/DN OTE N10:9/14 BND BND EOR
%   B30:0/11  PNEU_PX_IN_INST  "PX5 installed" %
%   N10:36  PNEU_PX_PSIG %
%   N7:68  LP_INT_PNEU_ALM_SP %
%   I:1.0/2  INT_PNEU_PRES_SWITCH  "PS-3" %
%   N10:0  SYSTEM_STATE  "STATE The current state of the system" %
%   N9:6  SYSTEM_PURGE %
%   B26:0/0  LP_INT_PNEU_ALM_EN %
%   T4:36  LP_INT_PNEU_ALM_TMR %
%   N10:7/14  LP_INT_PNEU_ALARM %
%   N7:69  LP_INT_PNEU_WRN_SP %
%   B26:5/0  LP_INT_PNEU_WRN_EN %
%   T4:37  LP_INT_PNEU_WRN_TMR %
%   N10:9/14  LP_INT_PNEU_WARN %

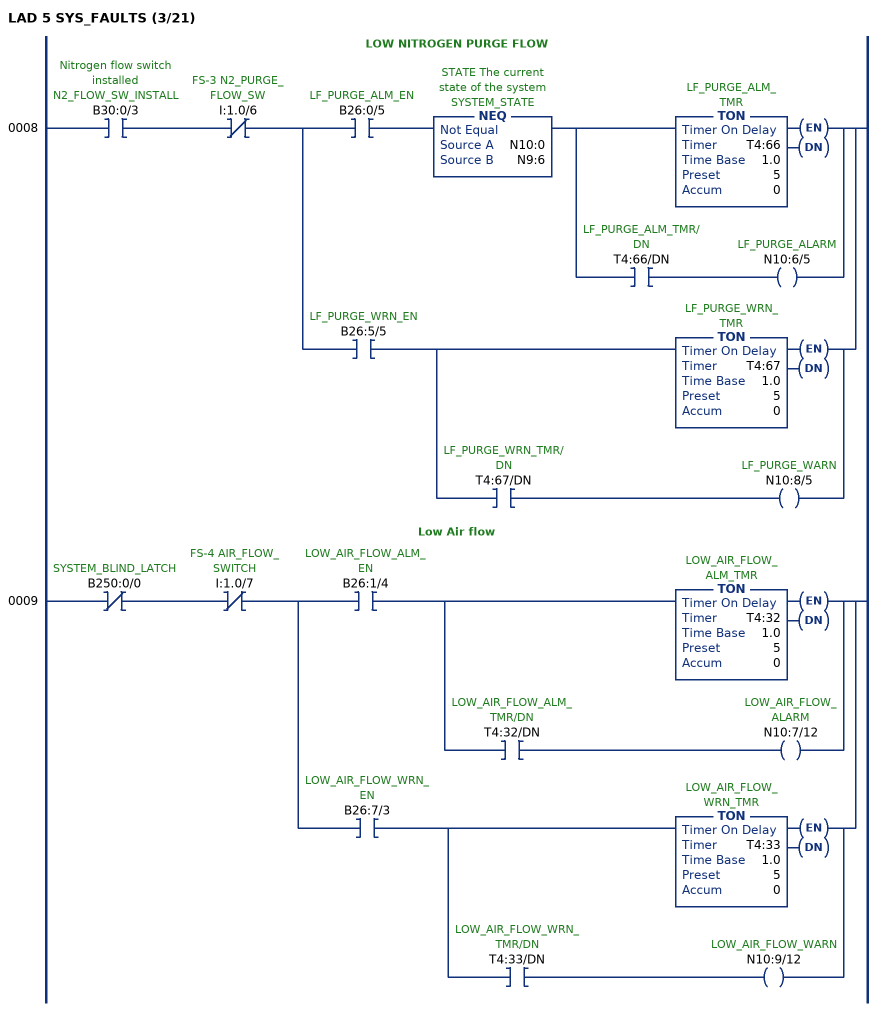
% Rung: 8 %
% TITLE: LOW NITROGEN PURGE FLOW %
SOR XIC B30:0/3 XIO I:1.0/6 BST XIC B26:0/5 NEQ N10:0 N9:6 BST TON T4:66 1.0 5 0 NXB XIC T4:66/DN OTE N10:6/5 BND NXB XIC B26:5/5 BST TON T4:67 1.0 5 0 NXB XIC T4:67/DN OTE N10:8/5 BND BND EOR
%   B30:0/3  N2_FLOW_SW_INSTALL  "Nitrogen flow switch installed" %
%   I:1.0/6  N2_PURGE_FLOW_SW  "FS-3" %
%   B26:0/5  LF_PURGE_ALM_EN %
%   N10:0  SYSTEM_STATE  "STATE The current state of the system" %
%   N9:6  SYSTEM_PURGE %
%   T4:66  LF_PURGE_ALM_TMR %
%   N10:6/5  LF_PURGE_ALARM %
%   B26:5/5  LF_PURGE_WRN_EN %
%   T4:67  LF_PURGE_WRN_TMR %
%   N10:8/5  LF_PURGE_WARN %
% Rung: 9 %
% TITLE: Low Air flow %
SOR XIO B250:0/0 XIO I:1.0/7 BST XIC B26:1/4 BST TON T4:32 1.0 5 0 NXB XIC T4:32/DN OTE N10:7/12 BND NXB XIC B26:7/3 BST TON T4:33 1.0 5 0 NXB XIC T4:33/DN OTE N10:9/12 BND BND EOR
%   B250:0/0  SYSTEM_BLIND_LATCH %
%   I:1.0/7  AIR_FLOW_SWITCH  "FS-4" %
%   B26:1/4  LOW_AIR_FLOW_ALM_EN %
%   T4:32  LOW_AIR_FLOW_ALM_TMR %
%   N10:7/12  LOW_AIR_FLOW_ALARM %
%   B26:7/3  LOW_AIR_FLOW_WRN_EN %
%   T4:33  LOW_AIR_FLOW_WRN_TMR %
%   N10:9/12  LOW_AIR_FLOW_WARN %

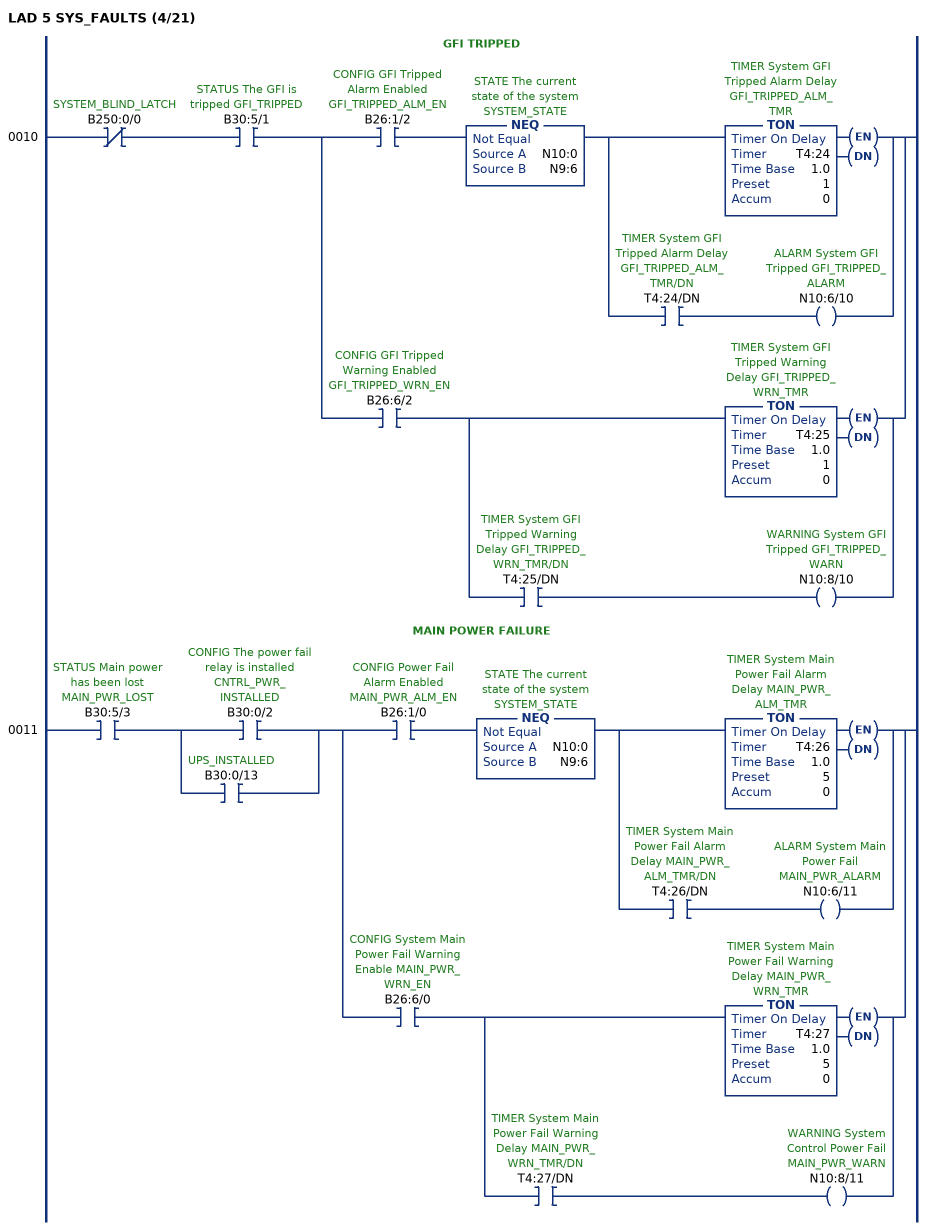
% Rung: 10 %
% TITLE: GFI TRIPPED %
SOR XIO B250:0/0 XIC B30:5/1 BST XIC B26:1/2 NEQ N10:0 N9:6 BST TON T4:24 1.0 1 0 NXB XIC T4:24/DN OTE N10:6/10 BND NXB XIC B26:6/2 BST TON T4:25 1.0 1 0 NXB XIC T4:25/DN OTE N10:8/10 BND BND EOR
%   B250:0/0  SYSTEM_BLIND_LATCH %
%   B30:5/1  GFI_TRIPPED  "STATUS The GFI is tripped" %
%   B26:1/2  GFI_TRIPPED_ALM_EN  "CONFIG GFI Tripped Alarm Enabled" %
%   N10:0  SYSTEM_STATE  "STATE The current state of the system" %
%   N9:6  SYSTEM_PURGE %
%   T4:24  GFI_TRIPPED_ALM_TMR  "TIMER System GFI Tripped Alarm Delay" %
%   N10:6/10  GFI_TRIPPED_ALARM  "ALARM System GFI Tripped" %
%   B26:6/2  GFI_TRIPPED_WRN_EN  "CONFIG GFI Tripped Warning Enabled" %
%   T4:25  GFI_TRIPPED_WRN_TMR  "TIMER System GFI Tripped Warning Delay" %
%   N10:8/10  GFI_TRIPPED_WARN  "WARNING System GFI Tripped" %
% Rung: 11 %
% TITLE: MAIN POWER FAILURE %
SOR XIC B30:5/3 BST XIC B30:0/2 NXB XIC B30:0/13 BND BST XIC B26:1/0 NEQ N10:0 N9:6 BST TON T4:26 1.0 5 0 NXB XIC T4:26/DN OTE N10:6/11 BND NXB XIC B26:6/0 BST TON T4:27 1.0 5 0 NXB XIC T4:27/DN OTE N10:8/11 BND BND EOR
%   B30:5/3  MAIN_PWR_LOST  "STATUS Main power has been lost" %
%   B30:0/2  CNTRL_PWR_INSTALLED  "CONFIG The power fail relay is installed" %
%   B30:0/13  UPS_INSTALLED %
%   B26:1/0  MAIN_PWR_ALM_EN  "CONFIG Power Fail Alarm Enabled" %
%   N10:0  SYSTEM_STATE  "STATE The current state of the system" %
%   N9:6  SYSTEM_PURGE %
%   T4:26  MAIN_PWR_ALM_TMR  "TIMER System Main Power Fail Alarm Delay" %
%   N10:6/11  MAIN_PWR_ALARM  "ALARM System Main Power Fail" %
%   B26:6/0  MAIN_PWR_WRN_EN  "CONFIG System Main Power Fail Warning Enable" %
%   T4:27  MAIN_PWR_WRN_TMR  "TIMER System Main Power Fail Warning Delay" %
%   N10:8/11  MAIN_PWR_WARN  "WARNING System Control Power Fail" %

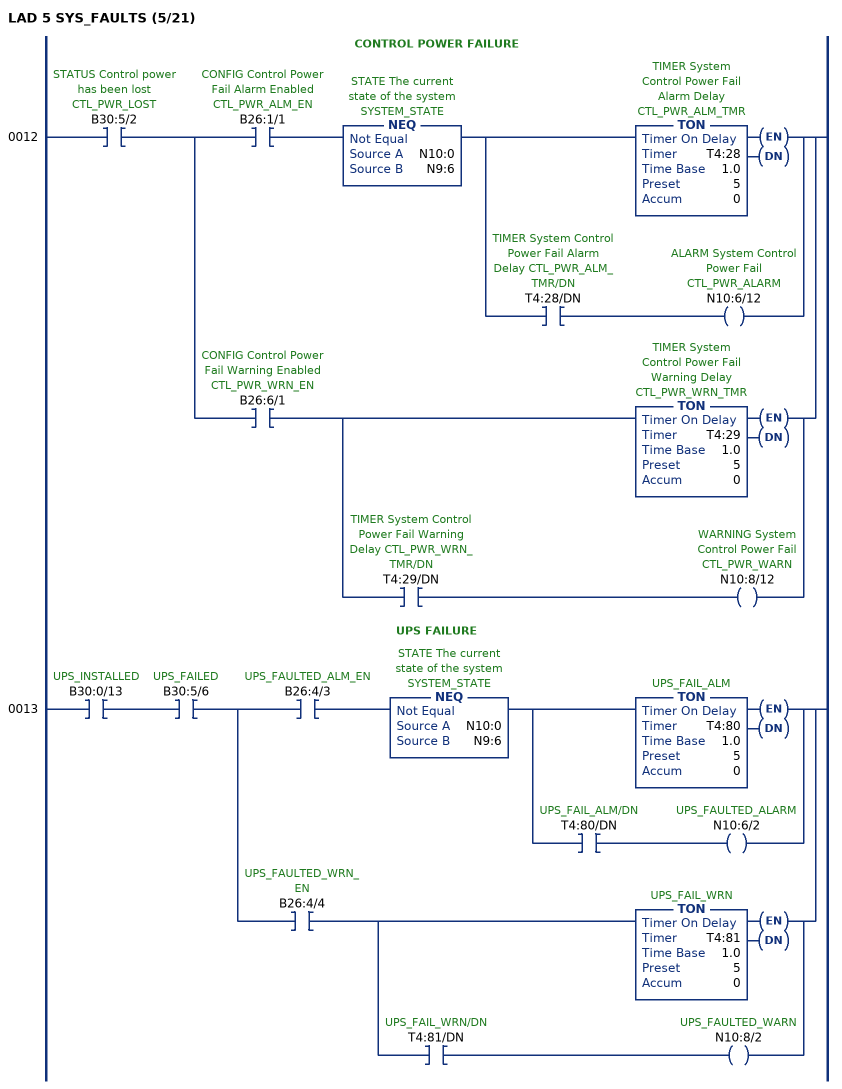
% Rung: 12 %
% TITLE: CONTROL POWER FAILURE %
SOR XIC B30:5/2 BST XIC B26:1/1 NEQ N10:0 N9:6 BST TON T4:28 1.0 5 0 NXB XIC T4:28/DN OTE N10:6/12 BND NXB XIC B26:6/1 BST TON T4:29 1.0 5 0 NXB XIC T4:29/DN OTE N10:8/12 BND BND EOR
%   B30:5/2  CTL_PWR_LOST  "STATUS Control power has been lost" %
%   B26:1/1  CTL_PWR_ALM_EN  "CONFIG Control Power Fail Alarm Enabled" %
%   N10:0  SYSTEM_STATE  "STATE The current state of the system" %
%   N9:6  SYSTEM_PURGE %
%   T4:28  CTL_PWR_ALM_TMR  "TIMER System Control Power Fail Alarm Delay" %
%   N10:6/12  CTL_PWR_ALARM  "ALARM System Control Power Fail" %
%   B26:6/1  CTL_PWR_WRN_EN  "CONFIG Control Power Fail Warning Enabled" %
%   T4:29  CTL_PWR_WRN_TMR  "TIMER System Control Power Fail Warning Delay" %
%   N10:8/12  CTL_PWR_WARN  "WARNING System Control Power Fail" %
% Rung: 13 %
% TITLE: UPS FAILURE %
SOR XIC B30:0/13 XIC B30:5/6 BST XIC B26:4/3 NEQ N10:0 N9:6 BST TON T4:80 1.0 5 0 NXB XIC T4:80/DN OTE N10:6/2 BND NXB XIC B26:4/4 BST TON T4:81 1.0 5 0 NXB XIC T4:81/DN OTE N10:8/2 BND BND EOR
%   B30:0/13  UPS_INSTALLED %
%   B30:5/6  UPS_FAILED %
%   B26:4/3  UPS_FAULTED_ALM_EN %
%   N10:0  SYSTEM_STATE  "STATE The current state of the system" %
%   N9:6  SYSTEM_PURGE %
%   T4:80  UPS_FAIL_ALM %
%   N10:6/2  UPS_FAULTED_ALARM %
%   B26:4/4  UPS_FAULTED_WRN_EN %
%   T4:81  UPS_FAIL_WRN %
%   N10:8/2  UPS_FAULTED_WARN %

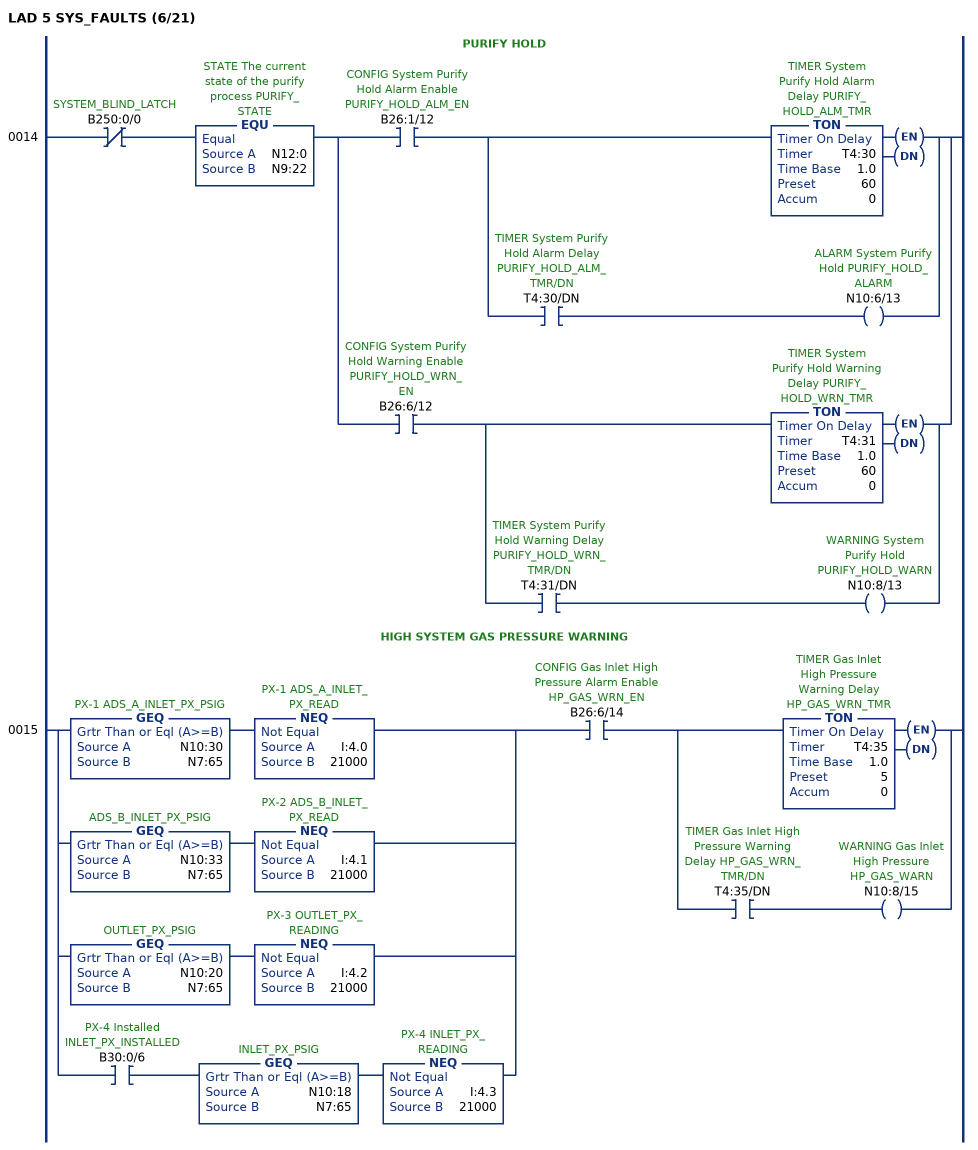
% Rung: 14 %
% TITLE: PURIFY HOLD %
SOR XIO B250:0/0 EQU N12:0 N9:22 BST XIC B26:1/12 BST TON T4:30 1.0 60 0 NXB XIC T4:30/DN OTE N10:6/13 BND NXB XIC B26:6/12 BST TON T4:31 1.0 60 0 NXB XIC T4:31/DN OTE N10:8/13 BND BND EOR
%   B250:0/0  SYSTEM_BLIND_LATCH %
%   N12:0  PURIFY_STATE  "STATE The current state of the purify process" %
%   N9:22  PURIFY_HOLD  "STATE Purify Hold" %
%   B26:1/12  PURIFY_HOLD_ALM_EN  "CONFIG System Purify Hold Alarm Enable" %
%   T4:30  PURIFY_HOLD_ALM_TMR  "TIMER System Purify Hold Alarm Delay" %
%   N10:6/13  PURIFY_HOLD_ALARM  "ALARM System Purify Hold" %
%   B26:6/12  PURIFY_HOLD_WRN_EN  "CONFIG System Purify Hold Warning Enable" %
%   T4:31  PURIFY_HOLD_WRN_TMR  "TIMER System Purify Hold Warning Delay" %
%   N10:8/13  PURIFY_HOLD_WARN  "WARNING System Purify Hold" %
% Rung: 15 %
% TITLE: HIGH SYSTEM GAS PRESSURE WARNING %
SOR BST GEQ N10:30 N7:65 NEQ I:4.0 21000 NXB GEQ N10:33 N7:65 NEQ I:4.1 21000 NXB GEQ N10:20 N7:65 NEQ I:4.2 21000 NXB XIC B30:0/6 GEQ N10:18 N7:65 NEQ I:4.3 21000 BND XIC B26:6/14 BST TON T4:35 1.0 5 0 NXB XIC T4:35/DN OTE N10:8/15 BND EOR
%   N10:30  ADS_A_INLET_PX_PSIG  "PX-1" %
%   N7:65  HP_GAS_WRN_SP  "CONFIG Gas Inlet High Pressure Warning Setpoint" %
%   I:4.0  ADS_A_INLET_PX_READ  "PX-1" %
%   N10:33  ADS_B_INLET_PX_PSIG %
%   I:4.1  ADS_B_INLET_PX_READ  "PX-2" %
%   N10:20  OUTLET_PX_PSIG %
%   I:4.2  OUTLET_PX_READING  "PX-3" %
%   B30:0/6  INLET_PX_INSTALLED  "PX-4 Installed" %
%   N10:18  INLET_PX_PSIG %
%   I:4.3  INLET_PX_READING  "PX-4" %
%   B26:6/14  HP_GAS_WRN_EN  "CONFIG Gas Inlet High Pressure Alarm Enable" %
%   T4:35  HP_GAS_WRN_TMR  "TIMER Gas Inlet High Pressure Warning Delay" %
%   N10:8/15  HP_GAS_WARN  "WARNING Gas Inlet High Pressure" %

